FUNCTION_BLOCK OF_E_TRAIN (* Generate of a finite train of events seperated by the time DT *)
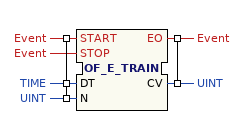
  EVENT_INPUT
    START WITH DT, N; (* Start event generation *)
    STOP; (* Stop event generation *)
  END_EVENT
  EVENT_OUTPUT
    EO WITH CV; (* Generated events *)
  END_EVENT
  VAR_INPUT
    DT : TIME; (* Time by which the events should be seperated *)
    N : UINT; (* Number of events to generate *)
  END_VAR
  VAR_OUTPUT
    CV : UINT; (* count of the current event: EO index (0..N-1) *)
  END_VAR
END_FUNCTION_BLOCK
